FUNCTION_BLOCK stubMover EXTENDS XtsMover
VAR
	stubTrack : XtsTrack('');
	iStubTrack : I_XtsTrack := stubTrack;
END_VAR

METHOD setAAbsPosition : HRESULT
VAR_INPUT
	setPos : LREAL;	
END_VAR
_MyNCData.ActPos := setPos;
END_METHOD

METHOD setActive : bool
VAR_INPUT
END_VAR
_myStatus.isActive := true;
END_METHOD

METHOD setAPosition : HRESULT
VAR_INPUT
	testPos : LREAL;
END_VAR
_stTmsActPositions.fTrackPosition := testPos;
_CurrentTrack := iStubTrack;
END_METHOD

METHOD setDisabled : HRESULT
VAR_INPUT
END_VAR
_MyAxisStatus.Disabled := true;
END_METHOD

METHOD setEnabled : HRESULT
VAR_INPUT
END_VAR
_MyAxisStatus.Disabled := false;
END_METHOD

METHOD setMoving
VAR_INPUT
END_VAR
_MyAxisStatus.NotMoving := FALSE;
END_METHOD

METHOD setNotActive : BOOL
VAR_INPUT
END_VAR
_myStatus.isActive := FALSE;
END_METHOD

METHOD setStationary
VAR_INPUT
END_VAR
_MyAxisStatus.NotMoving := TRUE;
END_METHOD

END_FUNCTION_BLOCK

(* stored: Version 1.1.0.1
   POU stubMover: Id {706dd25a-c636-4171-8a04-61e8c6b6cc8b}, SpecialFunc None
   Method setAAbsPosition: Id {387a1d1f-236f-462e-ac6c-91de4bc7f376}
   Method setActive: Id {d7d30cb6-d4e3-4284-903b-85caced60c68}
   Method setAPosition: Id {2798e35e-433b-437c-8074-09d525f98355}
   Method setDisabled: Id {3b4d37b1-2aff-4bc5-8d73-849300142d9c}
   Method setEnabled: Id {233db24b-81bf-4843-8554-24f39941731b}
   Method setMoving: Id {f76bd115-0fd7-43ee-a648-6fc15f420b4b}
   Method setNotActive: Id {06553b99-275a-43f9-b622-c0c80754e2f5}
   Method setStationary: Id {58cf9c7d-1727-4a74-b8f3-b9dc5225f246} *)
